{attribute 'GeneratedUsingTerminal: EP9128-0020-0016'}
{attribute addProperty BoxType "EP9128-0020-0016"}
{attribute addProperty Id "A_0004_EP9128_0021_0016A_0004_EP9128_0021_0016_3E1EBC3B589A_0001_EP9128_0020_0016_2_EP9128_1020EP9128_AB5A94672A_0001_EP9128_0020_0016_3_EP9128_2020EP9128_AB5A94672"}
{attribute addProperty CRC "1963361660"}
{attribute addProperty Size "593"}
TYPE A_0001_EP9128_0020_0016_7506857C EXTENDS EP9128_AB5A9467 :
STRUCT
	{attribute addProperty Name "A_0004_EP9128_0021_0016"}
	{attribute addProperty PreviousPort "A_0001(EP9128-0020-0016) : D"}
	A_0004_EP9128_0021_0016 : A_0004_EP9128_0021_0016_3E1EBC3B;
	{attribute addProperty Name "A_0001_EP9128_0020_0016_2_EP9128_1020"}
	{attribute addProperty PreviousPort "A_0001(EP9128-0020-0016) : C"}
	A_0001_EP9128_0020_0016_2_EP9128_1020 : EP9128_AB5A9467;
	{attribute addProperty Name "A_0001_EP9128_0020_0016_3_EP9128_2020"}
	{attribute addProperty PreviousPort "A_0001(EP9128-0020-0016)_2 (EP9128-1020) : C"}
	A_0001_EP9128_0020_0016_3_EP9128_2020 : EP9128_AB5A9467;
END_STRUCT
END_TYPE

(* stored: Version 1.2.0.0, ProductVersion 3.1.4024.9
   DUT A_0001_EP9128_0020_0016_7506857C: Id {13e08e16-e6df-4b68-9cfd-5d70b0f17ea2} *)
